// TIA Portal V20 export
// export: Created 2025-12-01T14:57:10.3744011Z, ExportSetting None, DisplayName Totally Integrated Automation Portal, DisplayVersion V20 Update 3, DisplayName TIA Portal Openness, DisplayVersion V20 Update 3, DisplayName TIA Portal Version Control Interface, DisplayVersion V20 Update 3, DisplayName STEP 7 Professional, DisplayVersion V20 Update 3, DisplayName STEP 7 Safety, DisplayVersion V20 Update 2, DisplayName WinCC Basic/Comfort/Advanced, DisplayVersion V20 Update 3, DisplayName WinCC Professional, DisplayVersion V20 Update 3, DisplayName WinCC Unified, DisplayVersion V20 Update 3
FUNCTION "FC820_EstadosDispositivos" : Void   // FC820, LAD
TITLE = "EstadosDispositivos" - Calcular los Eventos de los Dispositivos
{ S7_Optimized_Access := 'FALSE' }
AUTHOR : TRACKING
NAME : 20160407
VERSION : 4.1
// - Inicializar
// 
// - Bucle de Dispositivos CCPIF y CBOX
//   - Cierre del protocolo
//   - Calculo de los eventos de las presencias
//   - Calculo de los eventos generales
// 
// - Bucle de Disporisitivos Mesas
//   - Cierre del protocolo
//   - Calculo de los eventos de las presencias
//   - Calculo de los eventos generales
// 
// - Bucle de Disporisitivos Maquinas
//   - Cierre del protocolo
//   - Calculo de los eventos de las presencias
//   - Calculo de los eventos generales
// stored: AutoNumber false, SetENOAutomatically false
   VAR_TEMP
      EmiProtocoloDispositivoMesa : "UDT_ProtocoloEmiDispositivo";
      P_EmiProtocolo : DWord;
      NumeroMesa : UInt;   // Numero de Mesa Dispositivo
      MesaDeJDT02 : Bool;
      DispoDeJDT02 : Bool;
   END_VAR
BEGIN

NETWORK
TITLE = Inicializar
// Inicializacion de las variables de los DB's
/////////////////////////////////////////////////////////////////////////
// Inicializaciones de las variables de los DB's



NETWORK
TITLE = Bucle de los Dispositivos Mesas
// - Recorrer todos los dispositivos
//   - Mirar si ha cerrado el protocolo
//   - Mirar si hay algun evento de presencia
//   - Mirar si hay algun evento general
Bucle_DispositivoMesa:NOP   0;

/////////////////////////////////////////////////////////////////////////
//                        Recorrer todos las Mesas
/////////////////////////////////////////////////////////////////////////
// --- Inicializacion de los Punteros
// --- Recoger el WORD de Emision del Dispositivo
// --- Mirar si se ha cerrado el Protocolo del Dispositivo
// --- Recoger los datos del Dispositivo
// --- Mirar si hay algun Evento Pendiente por tratar (No debe haber ninguno)
// --- Mirar si se ha Activado alguna Presencia
// --- Mirar si hay alguna peticion pendiente (General)
// --- Si hay cambio de Estado el dispositivo
//

      L     1;
      T     #NumeroMesa;

/////////////////////////////////////////////////////////////////////////
// --- Inicializacin de los Punteros
InicioBucle_DispositivoMesa:NOP   0;

/////////////////////////////////////////////////////////////////////////
/// Mirar Si hay Mesa Configurada (2019 / 01 /18)
      SET;
      AN    "DB850_DefinicionMesas".Mesa[#NumeroMesa].ConfigMesa.MesaPaso;
      AN    "DB850_DefinicionMesas".Mesa[#NumeroMesa].ConfigMesa.MesaCruce;
      AN    "DB850_DefinicionMesas".Mesa[#NumeroMesa].ConfigMesa.MesaMultiplesDestinos;
      AN    "DB850_DefinicionMesas".Mesa[#NumeroMesa].ConfigMesa.MesaTL;
      JC    FinBucle_DispositivoMesa;


/////////////////////////////////////////////////////////////////////////
// --- Recoger Datos del Dispositivo (Protocolo)
      CALL  MOVE
      ( IN  := "DB840_Emision".DispoMesa[#NumeroMesa].Protocolo,
        OUT := #EmiProtocoloDispositivoMesa
      );

      L     P##EmiProtocoloDispositivoMesa;
      T     #P_EmiProtocolo;


/////////////////////////////////////////////////////////////////////////
// --- Recoger el Estado del Armari del Emision del Dispositivo
// --- Guardarlo en Real en la Base de Datos
//     Codigo de Error = ErrorReal
//     Bits de Estado

      L     "DB840_Emision".DispoMesa[#NumeroMesa].Error;
      T     "DB831_Mesas".Mesas[#NumeroMesa].ErrorReal;

      L     LW [#P_EmiProtocolo];
      L     W#16#7700;  // Solo la Parte Baja
      AW;
      SRD   8;
      T     "DB831_Mesas".Mesas[#NumeroMesa].StatusReal;


/////////////////////////////////////////////////////////////////////////
// --- Mirar si se ha cerrado el protocolo dl Dispositivo
      SET;
      L     "DB831_Mesas".Mesas[#NumeroMesa].EstadoPresenciaDispo;
      L     0;
      <>I;
      JC    CerrarProtocolo_DispositivoMesa;


/////////////////////////////////////////////////////////////////////////
// --- Mirar si hay algun Evento Pendiente por tratar (No debe haber ninguno)
//     * StatusRecepcion = 0
//     * StatusEmision = 0
      SET;
      L     "DB831_Mesas".Mesas[#NumeroMesa].EstadoRecepcionEvento;
      L     0;  // No hay nada, Eventos Recibidos
      <>I;
      JC    FinBucle_DispositivoMesa;

      SET;
      L     "DB831_Mesas".Mesas[#NumeroMesa].EstadoEmisionEvento;
      L     0;  // No hay nada, Eventos a Emitir
      <>I;
      JC    FinBucle_DispositivoMesa;


/////////////////////////////////////////////////////////////////////////
// --- Mirar si se ha Activado alguna Presencia

      L     LW [#P_EmiProtocolo];
      L     W#16#7F;  // Solo la Parte Alta
      AW;
      L     0;  // Mirar si se altivado algo ?
      <>I;
      JC    TratarPresencias_DispositivoMesa;


/////////////////////////////////////////////////////////////////////////
// --- Mirar si hay alguna peticion pendiente
      SET;
      L     "DB831_Mesas".Mesas[#NumeroMesa].EstadoGeneralEvento;
      L     0;  // No hay nada, Peticion Pendiente
      <>I;
      JC    TratarEstadoGeneral_DispositivoMesa;


/////////////////////////////////////////////////////////////////////////
// --- Si hay cambio de Estado el dispositivo
      SET;
      L     "DB831_Mesas".Mesas[#NumeroMesa].StatusReal;
      L     0;
      ==I;
      JC    FinBucle_DispositivoMesa;

      SET;
      L     "DB831_Mesas".Mesas[#NumeroMesa].StatusReal;
      L     "DB831_Mesas".Mesas[#NumeroMesa].StatusActual;
      ==I;  // Real = Actual (Guardado)
      JC    FinBucle_DispositivoMesa;


/////////////////////////////////////////////////////////////////////////
// --- Sin conexion no se genera el CAMBIO DE ESTADO (2019 01 18)
///    Mirar Si pertenece al JDT
      SET;
      A     "DB850_DefinicionMesas".Mesa[#NumeroMesa].ConfigMesa.MesaDeJDT02;  // JDT01 ?
      =     #MesaDeJDT02;

      SET;  // Esta Conectado ?
      AN    #MesaDeJDT02;  // Mirar Si esta el EnlaceCP Activo
      AN    "DB801_JDT01StatusCOM".EnlaceCP_OK;
      JC    FinBucle_DispositivoMesa;

      SET;  // Esta Conectado ?
      A     #MesaDeJDT02;  // Mirar Si esta el EnlaceCP Activo
      AN    "DB701_JDT02StatusCOM".EnlaceCP_OK;
      JC    FinBucle_DispositivoMesa;


/////////////////////////////////////////////////////////////////////////
// --- Guardo el nuevo estado y genero el evento
      L     "DB831_Mesas".Mesas[#NumeroMesa].StatusReal;
      T     "DB831_Mesas".Mesas[#NumeroMesa].StatusActual;
      L     "DB831_Mesas".Mesas[#NumeroMesa].ErrorReal;
      T     "DB831_Mesas".Mesas[#NumeroMesa].ErrorActual;

      L     160;  // 160 - Refresco de datos del Dispositivo
      T     "DB831_Mesas".Mesas[#NumeroMesa].EstadoEmisionEvento;


/////////////////////////////////////////////////////////////////////////
/////////////////////////////////////////////////////////////////////////
/////////////////////////////////////////////////////////////////////////
// --- Voy al siguiente Dispositivo
FinBucle_DispositivoMesa:NOP   0;
      L     #NumeroMesa;  // Incremento en 1 el Numero de Mesa
      L     1;
      +I;
      T     #NumeroMesa;

      L     #NumeroMesa;
      L     "CTE_MaxMesas";
      >I;  // Bucle de Maquinas
      JC    FinalFuncion;

/////////////////////////////////////////////////////////////////////////
// Finalizar, Siguiente Mesa
      JU    InicioBucle_DispositivoMesa;



NETWORK
TITLE = Cierre de Protocolo (Dispositivos) Mesas
// - Cierre de Protocolo del Dispositivo
//   * Fase 1 - Esperando que se desactive Emision del Dispositivo
CerrarProtocolo_DispositivoMesa:NOP   0;

/////////////////////////////////////////////////////////////////////////
/////////////////////////////////////////////////////////////////////////
/////////////////////////////////////////////////////////////////////////
// --- Cierre del protocolo del Dispositivo
//     * Esta en Fase 1 - Esperando que se desactive Emision del Dispositivo
      L     LW [#P_EmiProtocolo];
      L     W#16#7F;  // Solo la Parte Alta
      AW;
      L     0;  // Mirar si se altivado algo ?
      <>I;
      JC    FinCerrarProtocolo_DispositivoMesa;


/////////////////////////////////////////////////////////////////////////
// - Terminar Protocolo
      SET;  // DesActivar - EmiOK del dispositivo
      R     "DB841_Recepcion".DispoMesa[#NumeroMesa].Protocolo.EmiOK;

      L     0;  // Pasar a Fase 0, Acabado el Protocolo
      T     "DB831_Mesas".Mesas[#NumeroMesa].EstadoPresenciaDispo;

      JU    FinCerrarProtocolo_DispositivoMesa;


/////////////////////////////////////////////////////////////////////////
// - ReEscribir Protocolo
ReEscribirProtocolo_DispositivoMesa:NOP   0;
      SET;  // Activar - EmiOK del dispositivo
      S     "DB841_Recepcion".DispoMesa[#NumeroMesa].Protocolo.EmiOK;

      JU    FinCerrarProtocolo_DispositivoMesa;


/////////////////////////////////////////////////////////////////////////
/////////////////////////////////////////////////////////////////////////
/////////////////////////////////////////////////////////////////////////
// --- Final del Cierre del Protocolo del Dispositivo
FinCerrarProtocolo_DispositivoMesa:NOP   0;

// Finalizar, Siguiente Mesa
      JU    FinBucle_DispositivoMesa;



NETWORK
TITLE = Calculo de Eventos de las Presencias (Dispositivos) Mesas
// - Distribucion dependiendo del la presencia (Evento a Generar
//   * Evento de Reset OK
//   * Evento de Reset NOK
//   * Evento de Paro Blando OK
//   * Evento de Paro Blando NOK
// 
// - Empezar el cierre del protocolo
TratarPresencias_DispositivoMesa:NOP   0;

/////////////////////////////////////////////////////////////////////////
/////////////////////////////////////////////////////////////////////////
/////////////////////////////////////////////////////////////////////////
// --- Distribucion por las Presencias (Generar Evento correspondiente)
      SET;  // Evento de Reset OK
      A     #EmiProtocoloDispositivoMesa.ResetOK;
      JC    GenerarEventoResetOK_DispositivoMesa;

      SET;  // Evento de Reset NOK
      A     #EmiProtocoloDispositivoMesa.ResetNOK;
      JC    GenerarEventoResetNOK_DispositivoMesa;

      SET;  // Evento de ParoBlando OK
      A     #EmiProtocoloDispositivoMesa.ParoBlandoOK;
      JC    GenerarEventoParoBlandoOK_DispositivoMesa;

      SET;  // Evento de Paro Blando NOK
      A     #EmiProtocoloDispositivoMesa.ParoBlandoNOK;
      JC    GenerarEventoParoBlandoNOK_DispositivoMesa;


/////////////////////////////////////////////////////////////////////////
// --- No hay mas tipos de presencias programadas - cerrar el protocolo
//     Por defecto
      JU    DefectoTratarPresencias_DispositivoMesa;




/////////////////////////////////////////////////////////////////////////
/////////////////////////////////////////////////////////////////////////
/////////////////////////////////////////////////////////////////////////
// --- Generar Evento de Reset OK
// --- Empezar el cierre del Protocolo
GenerarEventoResetOK_DispositivoMesa:NOP   0;
      L     151;  // 151 - Reset OK del Dispositivo
      T     "DB831_Mesas".Mesas[#NumeroMesa].EstadoEmisionEvento;

      SET;  // Activar - EmiOK del dispositivo
      S     "DB841_Recepcion".DispoMesa[#NumeroMesa].Protocolo.EmiOK;

      L     1;  // Pasar a Fase 1, Empieza el Protocolo
      T     "DB831_Mesas".Mesas[#NumeroMesa].EstadoPresenciaDispo;

/////////////////////////////////////////////////////////////////////////
// Finalizar, Siguiente Dispositivo
      JU    FinBucle_DispositivoMesa;


/////////////////////////////////////////////////////////////////////////
/////////////////////////////////////////////////////////////////////////
/////////////////////////////////////////////////////////////////////////
// --- Generar Evento de Reset NOK
// --- Empezar el cierre del Protocolo
GenerarEventoResetNOK_DispositivoMesa:NOP   0;
      L     152;  // 152 - Reset NOK del Dispositivo
      T     "DB831_Mesas".Mesas[#NumeroMesa].EstadoEmisionEvento;

      SET;  // Activar - EmiOK del dispositivo
      S     "DB841_Recepcion".DispoMesa[#NumeroMesa].Protocolo.EmiOK;

      L     1;  // Pasar a Fase 1, Empieza el Protocolo
      T     "DB831_Mesas".Mesas[#NumeroMesa].EstadoPresenciaDispo;

/////////////////////////////////////////////////////////////////////////
// Finalizar, Siguiente Dispositivo
      JU    FinBucle_DispositivoMesa;


/////////////////////////////////////////////////////////////////////////
/////////////////////////////////////////////////////////////////////////
/////////////////////////////////////////////////////////////////////////
// --- Generar Evento de Paro Blando OK
// --- Empezar el cierre del Protocolo
GenerarEventoParoBlandoOK_DispositivoMesa:NOP   0;
      L     153;  // 153 - Paro Blando OK del Dispositivo
      T     "DB831_Mesas".Mesas[#NumeroMesa].EstadoEmisionEvento;

      SET;  // Activar - EmiOK del dispositivo
      S     "DB841_Recepcion".DispoMesa[#NumeroMesa].Protocolo.EmiOK;

      L     1;  // Pasar a Fase 1, Empieza el Protocolo
      T     "DB831_Mesas".Mesas[#NumeroMesa].EstadoPresenciaDispo;

/////////////////////////////////////////////////////////////////////////
// Finalizar, Siguiente Dispositivo
      JU    FinBucle_DispositivoMesa;


/////////////////////////////////////////////////////////////////////////
/////////////////////////////////////////////////////////////////////////
/////////////////////////////////////////////////////////////////////////
// --- Generar Evento de Paro Blando NOK
// --- Empezar el cierre del Protocolo
GenerarEventoParoBlandoNOK_DispositivoMesa:NOP   0;
      L     154;  // 154 - Paro Blando NOK del Dispositivo
      T     "DB831_Mesas".Mesas[#NumeroMesa].EstadoEmisionEvento;

      SET;  // Activar - EmiOK del dispositivo
      S     "DB841_Recepcion".DispoMesa[#NumeroMesa].Protocolo.EmiOK;

      L     1;  // Pasar a Fase 1, Empieza el Protocolo
      T     "DB831_Mesas".Mesas[#NumeroMesa].EstadoPresenciaDispo;

/////////////////////////////////////////////////////////////////////////
// Finalizar, Siguiente Dispositivo
      JU    FinBucle_DispositivoMesa;


/////////////////////////////////////////////////////////////////////////
/////////////////////////////////////////////////////////////////////////
/////////////////////////////////////////////////////////////////////////
// --- Empezar el cierre del Protocolo
DefectoTratarPresencias_DispositivoMesa:NOP   0;
      SET;  // Activar - EmiOK del dispositivo
      S     "DB841_Recepcion".DispoMesa[#NumeroMesa].Protocolo.EmiOK;

      L     1;  // Pasar a Fase 1, Empieza el Protocolo
      T     "DB831_Mesas".Mesas[#NumeroMesa].EstadoPresenciaDispo;

/////////////////////////////////////////////////////////////////////////
// Finalizar, Siguiente Dispositivo
      JU    FinBucle_DispositivoMesa;



NETWORK
TITLE = Calculo del Evento General (Dispositivos) Mesa
// - Distribucion de los eventos generales
//   * Refresco de datos del dispositivo
TratarEstadoGeneral_DispositivoMesa:NOP   0;

/////////////////////////////////////////////////////////////////////////
/////////////////////////////////////////////////////////////////////////
/////////////////////////////////////////////////////////////////////////
// --- Distribucion del evento general
      L     "DB831_Mesas".Mesas[#NumeroMesa].EstadoGeneralEvento;
      L     25;  // Peticion de Refescom de Datos
      ==I;
      JC    RefrescoDatos_EstadoGeneral_DispositivoMesa;

// --- No hay más programados
      JU    FinTratarEstadoGeneral_DispositivoMesa;


/////////////////////////////////////////////////////////////////////////
/////////////////////////////////////////////////////////////////////////
// --- Generar Evento de Refesco de Datos del Dispositivo
RefrescoDatos_EstadoGeneral_DispositivoMesa:NOP   0;
      L     "DB831_Mesas".Mesas[#NumeroMesa].StatusReal;
      T     "DB831_Mesas".Mesas[#NumeroMesa].StatusActual;
      L     "DB831_Mesas".Mesas[#NumeroMesa].ErrorReal;
      T     "DB831_Mesas".Mesas[#NumeroMesa].ErrorActual;

      SET;
      L     "DB831_Mesas".Mesas[#NumeroMesa].StatusActual;
      L     0;
      ==I;
      JC    NoExisteRefrescoDatos_EstadoGeneral_DispositivoMesa;

      L     160;  // 160 - Refresco de datos del Dispositivo
      T     "DB831_Mesas".Mesas[#NumeroMesa].EstadoEmisionEvento;


NoExisteRefrescoDatos_EstadoGeneral_DispositivoMesa:NOP   0;
      L     0;  // EstadoGeneral - Dar por Tratado
      T     "DB831_Mesas".Mesas[#NumeroMesa].EstadoGeneralEvento;

      JU    FinTratarEstadoGeneral_DispositivoMesa;


/////////////////////////////////////////////////////////////////////////
/////////////////////////////////////////////////////////////////////////
// --- Fin  de Eventos Generales
// Finalizar, Siguiente Dispositivo
FinTratarEstadoGeneral_DispositivoMesa:NOP   0;
      JU    FinBucle_DispositivoMesa;



NETWORK
TITLE = Finalizar
// Se Acabo
FinalFuncion:NOP   0;

END_FUNCTION
